FUNCTION_BLOCK ZAppSequenceBoot EXTENDS ZAppSequence IMPLEMENTS ZCore.ISequence
VAR
  _step : ZCore.Step(ZAppStep.BootBegin, ZAppStep.BootEnd);
END_VAR

IF OnStart(_step)
THEN
  // init custom sequence variables here ...
END_IF

REPEAT
  LogStep();

  CASE _step.Index OF
    (* -------------------------------------------------------------------------------------------------------------------------------- *)
    ZAppStep.BootBegin:
    (* -------------------------------------------------------------------------------------------------------------------------------- *)
    
      IF _step.OnEntry()
      THEN
        ZModuleProgram.LoggerFile.SetLevel(ZCore.LogLevel.Trace);
        ZModuleProgram.Logger.AddLogger(ZModuleProgram.LoggerFile);        
        {attribute '__ZwPlcAppZComModuleContext__'} // Do not remove this attribute! It is used for code generation.      
      END_IF
      
	  IF ZModuleProgram.Datetime.State <> ZCore.ObjectState.Booting
      THEN
        _step.SetNext(ZAppStep.BootLoadDefaultData);        
      END_IF
      
    (* -------------------------------------------------------------------------------------------------------------------------------- *)
    ZAppStep.BootLoadDefaultData:
    (* -------------------------------------------------------------------------------------------------------------------------------- *)

      {warning 'The application is loading the default config data on every restart!'}
      LoadDefaultConfigData();
      
      IF IsCommissioning()
      THEN
        LoadDefaultData();
      END_IF
      
      _step.SetNext(ZAppStep.BootEnd);
      
    (* -------------------------------------------------------------------------------------------------------------------------------- *)
    ZAppStep.BootEnd:
    (* -------------------------------------------------------------------------------------------------------------------------------- *)
      SetBusy(FALSE);
      
  ELSE
    Abort('sequence contains unhandled step');
  END_CASE
UNTIL _step.IsNotRepeatable() OR_ELSE NOT Busy END_REPEAT

METHOD  IsCommissioning : BOOL
IsCommissioning := TRUE;
END_METHOD

METHOD FINAL LoadDefaultConfigData

{region "Scribly"}
  {IF NOT (defined (Scribly_disabled))}
  ZGlobal.Data.Config.Scribly.Simulated := TRUE;
  {region "UserInitCode"}
  // put your individual init code for this unit here
  {endregion}
  {END_IF}
  {attribute 'ZId' := '61e5b130-0fef-4d8b-85dd-afb1efcde47c'}
{endregion}

{attribute '__ZwPlcUnitLoadDefaultConfigData__'} // Do not remove this attribute! It is used for code generation.
END_METHOD

METHOD FINAL LoadDefaultData

{attribute '__ZwPlcUnitLoadDefaultData__'} // Do not remove this attribute! It is used for code generation.
ZGlobal.Data.Machine.Scribly.Highspeed := 100;
ZGlobal.Data.Machine.Scribly.Slowspeed := 10;
END_METHOD

END_FUNCTION_BLOCK

(* stored: Version 1.1.0.1
   POU ZAppSequenceBoot: Id {4175e36d-67a3-44c7-aa0a-3e8bf9b3c409}, SpecialFunc None
   Method IsCommissioning: Id {a3ea03ec-ee5f-4d37-b289-be135ee49366}
   Method LoadDefaultConfigData: Id {033f4bff-60a4-468c-8813-fef0ea28cd35}
   Method LoadDefaultData: Id {fa9633c4-76dc-4ebb-990b-7115ef78f212} *)
